Fanuc KAREL source: ka00145.KL

-- PROVISIONAL review KL for V940-1; original PC SHA256 23aa3c0df0a9b1c6c5a751e5e54d361ccac9fdc12f61ffcebe3eceec76ae7476
-- Incomplete behavior may be omitted. Consult companion uncertainty JSON. Do not deploy.
PROGRAM KA00145
%NOLOCKGROUP
-- UNRESOLVED_DECL SRC type=002010
-- UNRESOLVED_DECL DST type=002010
BEGIN
  -- V9_COMPOSED_GLOBAL_TRANSFER_HINT repetitions=1; address IDs observed; pairing/direction/source/runtime held
  -- V9_TWO_GLOBAL_ADDRESS_COPY_HINT bounded five-record physical form; type/direction/source/runtime held
  -- V9_ZERO_TABLE_METADATA_HINT layout=0001; no indexed target words; source/name/runtime held
  -- UNRESOLVED_PC offsets 5-19; opcodes 22,22,1E
  -- UNRESOLVED_PC offsets 24-28; opcodes 7F
END KA00145
